{attribute 'no_check'}
FUNCTION_BLOCK EcFcDS402_ParkerAC30 EXTENDS EcFcDS402_ComBase IMPLEMENTS I_ActuatorFwdRev
VAR_INPUT
	RefVelo													: 	LREAL := 2000; 	//sets speed of rotation	
	RampUp											AT  %Q*	:	TIME := T#10S;	//0486: Acceleration Time
	RampDown										AT  %Q*	:	TIME := T#10S;	//0487: Deceleration Time
END_VAR                     							
VAR_OUTPUT               
	CiA_Control												:	CiA_DS402Controlword_Parker;
	CiA_Status												:	CiA_DS402Statusword_Parker;

	{attribute 'displaymode':='hex'}   							
	WarningCode										AT  %I*	:	UDINT;			//0829: Warnings  1 - 32
	ActVelo											AT  %I* : 	REAL; 			//0395: Actual Speed Percent
	Power											AT  %I*	: 	REAL; 			//0380: Power kW
	Q_TargetVelo							 	AT  %Q* :	REAL;			//0681: Comms Reference
END_VAR                 							
VAR (* IO Internal *)   							
END_VAR                 								
VAR                     	
END_VAR

(* Com Parker AC30 										V1.0   *)
(***************************************************************)

(* Protection Switch *******************************************)		
	IF ResetTrig  
	THEN 
		REset(); 
	END_IF
	
	ProtSwitchOK();	
	FuseBrakeOK(); (* same parameter like ProtSwitch *)

(* Contactor ***************************************************)
	Q_Contactor 											:= Contactor AND ProtSwitchOK.Q AND FuseBrakeOK.Q;

(* Read status *************************************************)
	CiA_Status.readStatusword(Statusword);

(* interpret status word ***************************************)
	Ready													:= CiA_Status.ReadyToSwitchOn AND Q_Contactor;
	Error													:= CiA_Status.Fault AND Q_Contactor;                       									
	Busy													:= CiA_Status.OperationEnabled AND ActVelo <> 0; 
	                                        
// write contorlword DS 402  ****************************************
	CiA_Control.SwitchOn									:= Enable AND Q_Contactor;
	CiA_Control.EnableOperation								:= FeedBwd AND StartBwd AND NOT Start OR Feed AND Start AND NOT StartBwd;
	CiA_Control.FaultReset									:= ResetIntern;
	CiA_Control.EnableRevOp									:= CiA_Control.EnableOperation AND 	StartBwd;						

(* setvalue ***************************************************)
	IF CiA_Control.EnableOperation AND RefVelo <> 0.0
	THEN
		IF StartBwd
		THEN
			Q_TargetVelo 									:= TO_REAL(Velo/RefVelo * 100.0  * -1); (* 1 Digit = 1 rpm *)
		ELSE	
			Q_TargetVelo									:= TO_REAL(Velo/RefVelo * 100.0); (* 1 Digit = 1 rpm *)
		END_IF	
	ELSE
		Q_TargetVelo										:= 0;
	END_IF
	
// Reset FALSE ****************************************************
	ResetIntern												:= FALSE;
	
(* HmiStatus **************************************************)
	Status.0 												:= CiA_Status.OperationEnabled AND StartBwd; 	// counter-clockwise rotation
	Status.1 												:= CiA_Status.OperationEnabled AND Start; 	// clockwise rotation
	Status.2 												:= ActVelo < 0;
	Status.3												:= ActVelo > 0;
	Status.4 												:= FeedBwd;
	Status.5 												:= Feed;
	Status.6 												:= Ready;
	Status.7 												:= Error;
// ****************************************************************

{attribute 'monitoring' := 'call'}
PROPERTY public forwardStarted : BOOL
GET
forwardStarted := CiA_Control.EnableOperation and Q_TargetVelo > 0;
END_GET
END_PROPERTY

{attribute 'monitoring' := 'call'}
PROPERTY public isDisabled : BOOL
GET
isDisabled := not CiA_Status.SwitchedOn and not CiA_Status.OperationEnabled;
END_GET
END_PROPERTY

{attribute 'monitoring' := 'call'}
PROPERTY public isEnabled : BOOL
GET
isEnabled := CiA_Status.SwitchedOn or CiA_Status.OperationEnabled;
END_GET
END_PROPERTY

{attribute 'monitoring' := 'call'}
PROPERTY public isOff : BOOL
GET
isOff := NOT CiA_Status.OperationEnabled;
END_GET
END_PROPERTY

{attribute 'monitoring' := 'call'}
PROPERTY public isOn : BOOL
GET
isOn := CiA_Status.OperationEnabled;
END_GET
END_PROPERTY

{attribute 'monitoring' := 'call'}
PROPERTY public reverseStarted : BOOL
GET
reverseStarted := CiA_Control.EnableOperation and Q_TargetVelo < 0;
END_GET
END_PROPERTY

METHOD setDisable : BOOL
VAR_INPUT
END_VAR

SetDisable													:= Super^.setDisable() AND NOT CiA_Status.SwitchedOn;
END_METHOD

METHOD setEnable : BOOL
VAR_INPUT
END_VAR

SetEnable													:= SUPER^.setEnable() AND CiA_Status.SwitchedOn;
END_METHOD

METHOD PUBLIC startForward : bool //Return busy flag
VAR_INPUT
END_VAR
Start 														:= TRUE; 
StartBwd 													:= FALSE;
startForward												:= Busy and Q_TargetVelo > 0;
END_METHOD

METHOD PUBLIC startReverse : bool //Return busy flag
VAR_INPUT
END_VAR
Start 														:= FALSE; 
StartBwd 													:= TRUE;
startReverse												:= Busy and Q_TargetVelo < 0;
END_METHOD

METHOD PUBLIC switchOn : BOOL  //True if motor is switched on
VAR_INPUT
END_VAR
switchOn := startForward();
END_METHOD

END_FUNCTION_BLOCK

(* stored: Version 1.1.0.1, ProductVersion 3.1.4024.13
   POU EcFcDS402_ParkerAC30: Id {abc6ca9c-9164-4f6c-abfa-e70e794f6326}, SpecialFunc None
   Folder methods: Id {0f7732c7-a54a-4f5a-87e1-4a2281ebcdf7}
   Folder properties: Id {f7668a6e-ebc6-4f42-8abb-8a3cc76a3f47}
   Property forwardStarted: Id {48f68d5b-e6ff-4256-8131-9767a5a70b6a}
   Get Get: Id {4663d6b5-d645-4a69-ad6f-316b20700ff8}
   Property isDisabled: Id {28f0547b-3488-4ec8-8d8d-3a7360d602ac}
   Get Get: Id {0a6d4449-7dfb-4cc6-bd54-3d8e6641a98a}
   Property isEnabled: Id {43ec42d4-f522-4731-9032-feeeb6841e18}
   Get Get: Id {3906fe97-a26b-44f8-9a83-900d44767882}
   Property isOff: Id {bbf0bec5-ff67-442b-b9bf-7634006874ce}
   Get Get: Id {f26f5183-ff4c-4dc4-8f72-a594fb39d246}
   Property isOn: Id {83171d3e-a27e-4bb3-97b3-b7589faba185}
   Get Get: Id {52067bc2-5713-41fd-8e02-dd716d369a91}
   Property reverseStarted: Id {6354b634-e07c-4dfd-af03-ee73ab16c05e}
   Get Get: Id {46549679-62f1-4b49-93bb-4335c73d1b4f}
   Method setDisable: Id {b3d78416-f239-48f5-b600-2631a3b1a421}
   Method setEnable: Id {680a0364-3574-4b0c-807f-f3ab962005c1}
   Method startForward: Id {d5776931-40b6-486e-a909-ce7346f307e1}
   Method startReverse: Id {f15f9d8d-2fa3-42d5-afe6-e6879d25eb51}
   Method switchOn: Id {8d2376b2-b2a0-4e45-af2f-6ac0b157e4eb} *)
